(* POU Mio_GetCardMode, IL *)
(******************************************************************************
Description: Gets the mode of an IO-card.
Input:
  - CardId: ID of the card
Return: 
  - MIO_RETSTATE.RetCode: DINT => Success- or error code
  - MIO_RETSTATE.State: DWORD =>  Card mode (valid in case of success)
******************************************************************************)
FUNCTION Mio_GetCardMode : MIO_RETSTATE
VAR_INPUT
	CardId: DINT;
END_VAR
LD 0
END_FUNCTION

(* POU Mio_GetChanInf, IL *)
(******************************************************************************
Description: Gets information of an IO-channel of a card
Input:
  - CardId: ID of the card
  - Chan: Channel number
Return: 
  - MIO_RETCHANINF.RetCode: DINT => Success- or error-code
  - MIO_RETCHANINF.ChanCategory: DWORD =>  Channel-category (valid in case of success)
  - MIO_RETCHANINF.ChanFlags: DWORD =>  Properies of channel (valid in case of success)
******************************************************************************)
FUNCTION Mio_GetChanInf : MIO_RETCHANINF
VAR_INPUT
	CardId: DINT;
	Chan: DINT;
END_VAR
LD 0
END_FUNCTION

(* POU Mio_GetChanMode, IL *)
(******************************************************************************
Description: Gets the mode of a channel of an IO-card.
Input:
  - CardId: ID of the card
  - Chan: Channel number
Return: 
  - MIO_RETSTATE.RetCode: DINT => Success- or error-code
  - MIO_RETSTATE.State: DWORD =>  Channel mode (valid in case of success)
******************************************************************************)
FUNCTION Mio_GetChanMode : MIO_RETSTATE
VAR_INPUT
	CardId: DINT;
	Chan: DINT;
END_VAR
LD 0
END_FUNCTION

(* POU Mio_GetChanRangeInf, ST *)
(******************************************************************************
Description: Gets range information of an IO-channel of a card
Input:
  - CardId: ID of the card
  - Chan: Channel number
Return: 
  - MIO_RETCHANINF.RetCode: DINT => Success- or error-code
  - MIO_RETCHANINF.ChanCategory: DWORD =>  Channel-category (valid in case of success)
  - MIO_RETCHANINF.ChanFlags: DWORD =>  Properies of channel (valid in case of success)
******************************************************************************)
FUNCTION Mio_GetChanRangeInf : MIO_RETCHANRANGEINF
VAR_INPUT
	CardId: DINT;
	Chan: DINT;
END_VAR
;
END_FUNCTION

(* POU MIO_GetCustomerID, ST *)
FUNCTION_BLOCK MIO_GetCustomerID
VAR_INPUT
	Req : BOOL;
	CardId: DINT;
	CryptoKey: UDINT;
	AlgorithmId: UDINT;
	UserData: UDINT;
	CryptoFn: STRING(255);
END_VAR
VAR_OUTPUT
	Done : BOOL;
	Error : BOOL;
	Status : DINT;
	CustomerID: UDINT;
END_VAR
VAR
	Pltd : DWORD;
END_VAR
;
END_FUNCTION_BLOCK

(* POU Mio_GetError, IL *)
(******************************************************************************
Description: Gets the error state of a channel of an IO-card
Input:
  - CardId: ID of the card
  - Chan: Channel number
Return: 
  - MIO_RETSTATE.RetCode: DINT => Success- or error code
  - MIO_RETSTATE.State: DWORD =>  Error state (valid in case of success)
******************************************************************************)
FUNCTION Mio_GetError : MIO_RETSTATE
VAR_INPUT
	CardId: DINT;
	Chan: DINT;
END_VAR
LD 0
END_FUNCTION

(* POU Mio_GetExtCardInf, IL *)
(******************************************************************************
Description: Gets extended info for an IO-card
Input:
  - CardId: ID of the card
Return: 
  - MIO_RETEXTCARDINF.RetCode => Success- or error-code
  - MIO_RETEXTCARDINF.CardNb => Card number
  - MIO_RETEXTCARDINF.StationNb => Station number
  - MIO_RETEXTCARDINF.SlotNb => Slot number
  - MIO_RETEXTCARDINF.PreSlots => Precessing-also-used-slots
  - MIO_RETEXTCARDINF.PostSlots => Following-also-used-slots
  - MIO_RETEXTCARDINF.Mode => Mode of card driver
  - MIO_RETEXTCARDINF.State => State of Card-Driver
  - MIO_RETEXTCARDINF.CardType => Card type
  - MIO_RETEXTCARDINF.CardVariant => Card variant
  - MIO_RETEXTCARDINF.CardCategory => Card category
  - MIO_RETEXTCARDINF.CardFlags => Properties of card
  - MIO_RETEXTCARDINF.MaxChan => Number of channels
  - MIO_RETEXTCARDINF.Version => Card version
  - MIO_RETEXTCARDINF.DrvVersion => Necc. driver version
  - MIO_RETEXTCARDINF.Attribute => Defined/set attributes
  - MIO_RETEXTCARDINF.ProdTime => Date + time of production
  - MIO_RETEXTCARDINF.ProdNb => Serial no.-string
  - MIO_RETEXTCARDINF.Name => Name of card
  - MIO_RETEXTCARDINF.Info => Block of info text
  - MIO_RETEXTCARDINF.DrvName => Name of driver-*.M file
  - MIO_RETEXTCARDINF.Power => Power consumption in [mW]
  - MIO_RETEXTCARDINF.Current_5V => 5V Current sink/source in [mA]
  - MIO_RETEXTCARDINF.Current_P15V => +15V Current sink/source in [mA]
  - MIO_RETEXTCARDINF.Current_M15V => -15V Current sink/source in [mA]
  - MIO_RETEXTCARDINF.ModVerType => Version Type code
  - MIO_RETEXTCARDINF.RedundantRead => Redundant read of data if TRUE
  - MIO_RETEXTCARDINF.WriteVerify => Write verify of data if TRUE
  - MIO_RETEXTCARDINF.BusCheck => BUSCHECK supported if TRUE
  - MIO_RETEXTCARDINF.AliveCheck => ALIVECHECK supported if TRUE
  - MIO_RETEXTCARDINF.AssemblyCode => Function code lower part
  - MIO_RETEXTCARDINF.HwVariant => Hardware variant
  - MIO_RETEXTCARDINF.Reserved1 => Not used, 0 for now
  - MIO_RETEXTCARDINF.Settings => Flags that may be en-/disabled
  - MIO_RETEXTCARDINF.Fware => Firmware version
  - MIO_RETEXTCARDINF.ExStateInfo => Extended state information


******************************************************************************)
FUNCTION Mio_GetExtCardInf : MIO_RETEXTCARDINF
VAR_INPUT
	CardId: DINT;			(* use special value 16#80000001 for 'Cpu-Card' *)
END_VAR
	LD		0
END_FUNCTION

(* POU Mio_GetExtCardInf2, ST *)
(******************************************************************************
Description: Gets extended info for an IO-card
Input:
  - CardId: ID of the card
Return: 
  - MIO_RETEXTCARDINF2.RetCode => Success- or error-code
  - MIO_RETEXTCARDINF2.CardNb => Card number
  - MIO_RETEXTCARDINF2.StationNb => Station number
  - MIO_RETEXTCARDINF2.SlotNb => Slot number
  - MIO_RETEXTCARDINF2.PreSlots => Precessing-also-used-slots
  - MIO_RETEXTCARDINF2.PostSlots => Following-also-used-slots
  - MIO_RETEXTCARDINF2.Mode => Mode of card driver
  - MIO_RETEXTCARDINF2.State => State of Card-Driver
  - MIO_RETEXTCARDINF2.CardType => Card type
  - MIO_RETEXTCARDINF2.CardVariant => Card variant
  - MIO_RETEXTCARDINF2.CardCategory => Card category
  - MIO_RETEXTCARDINF2.CardFlags => Properties of card
  - MIO_RETEXTCARDINF2.MaxChan => Number of channels
  - MIO_RETEXTCARDINF2.Version => Card version
  - MIO_RETEXTCARDINF2.DrvVersion => Necc. driver version
  - MIO_RETEXTCARDINF2.Attribute => Defined/set attributes
  - MIO_RETEXTCARDINF2.ProdTime => Date + time of production
  - MIO_RETEXTCARDINF2.ProdNb => Serial no.-string
  - MIO_RETEXTCARDINF2.Name => Name of card
  - MIO_RETEXTCARDINF2.Info => Block of info text
  - MIO_RETEXTCARDINF2.DrvName => Name of driver-*.M file
  - MIO_RETEXTCARDINF2.Power => Power consumption in [mW]
  - MIO_RETEXTCARDINF2.Current_5V => 5V Current sink/source in [mA]
  - MIO_RETEXTCARDINF2.Current_P15V => +15V Current sink/source in [mA]
  - MIO_RETEXTCARDINF2.Current_M15V => -15V Current sink/source in [mA]
  - MIO_RETEXTCARDINF2.ModVerType => Version Type code
  - MIO_RETEXTCARDINF2.RedundantRead => Redundant read of data if TRUE
  - MIO_RETEXTCARDINF2.WriteVerify => Write verify of data if TRUE
  - MIO_RETEXTCARDINF2.BusCheck => BUSCHECK supported if TRUE
  - MIO_RETEXTCARDINF2.AliveCheck => ALIVECHECK supported if TRUE
  - MIO_RETEXTCARDINF2.AssemblyCode => Function code lower part
  - MIO_RETEXTCARDINF2.HwVariant => Hardware variant
  - MIO_RETEXTCARDINF2.Reserved1 => Not used, 0 for now
  - MIO_RETEXTCARDINF2.Settings => Flags that may be en-/disabled
  - MIO_RETEXTCARDINF2.ExStateInfo => Extended state information
  - MIO_RETEXTCARDINF2.Versions => Versions of this module (FW, Logic, ...)
  - MIO_RETEXTCARDINF2.PackageVers => Package version
  - MIO_RETEXTCARDINF2.PartNumber => Part number (0 if not available)
  - MIO_RETEXTCARDINF2.FirmBackup => Firmware can be recovered
  - MIO_RETEXTCARDINF2.Spare1 => Align it to 32 bit
  - MIO_RETEXTCARDINF2.Spare => Not used, 0 for now

******************************************************************************)
FUNCTION Mio_GetExtCardInf2 : MIO_RETEXTCARDINF2
VAR_INPUT
	CardId: DINT;			(* use special value 16#80000001 for 'Cpu-Card' *)
END_VAR
;
END_FUNCTION

(* POU Mio_GetIdToCard, IL *)
(******************************************************************************
Description: Gets the ID of an IO-card specified by card number
Input:
  - CardNum: Number of the card
Return: 
  - DINT => Pointer-ID of Card
  - In case of error: the special value -2147483648 (16#80000000) is returned
******************************************************************************)
FUNCTION Mio_GetIdToCard : DINT
VAR_INPUT
	CardNum : DINT;
END_VAR
LD 0
END_FUNCTION

(* POU Mio_GetInterruptInfo, ST *)
(******************************************************************************
Description: Returns informations regarding the current interrupt cycle(Is only
    valid if the current project is configured to be interrupt triggered-Event
    or Error interrupt.)
Input:
  - Dummy: 
Return: 
  -
******************************************************************************)
FUNCTION Mio_GetInterruptInfo : MIO_INTINFO
VAR_INPUT
	Dummy: DINT;
END_VAR
;
END_FUNCTION

(* POU Mio_GetNewSlaveReboot, ST *)
(******************************************************************************
Description: Returns the configuration for new FAST Bus slave stations behaviour.
Input:
  - Dummy: 
Return: 
  - TRUE: The controller will reboot, as soon as a new station is recognized.
  - FALSE: The new station will not be usable until a reboot happens. 
******************************************************************************)
FUNCTION Mio_GetNewSlaveReboot : BOOL
VAR_INPUT
	Dummy: DINT;
END_VAR
;
END_FUNCTION

(* POU Mio_GetNextError, IL *)
(******************************************************************************
Description: Finds the next IO-card / channel with an error state with attention to
Input:
  - StartCard:  Card to start the search from, valid range starts with -1 
  - StartChan:  Chan to start the search from, valid range starts with -1 
  - CardId: ID of the card
  - Chan: Channel number
Return: 
  - MIO_RETFOUND.RetCode: DINT => Success (0 or 1) - or error-code (<0)
  - MIO_RETFOUND.Card: DINT =>  Card with error (-1 for none)  (valid in case of success)
  - MIO_RETFOUND.Chan: DINT =>   Chan with error (-1 for none) (valid in case of success)
  - MIO_RETFOUND.State: DWORD =>  Error state (valid in case of success)
******************************************************************************)
FUNCTION Mio_GetNextError : MIO_RETFOUND
VAR_INPUT
	StartCard: DINT;		(* Card to start the search from, valid range starts with -1 *)
	StartChan: DINT;		(* Chan to start the search from, valid range starts with -1 *)
END_VAR
LD 0
END_FUNCTION

(* POU Mio_GetPackedValues, ST *)
(******************************************************************************
Description: Gets a number of packed values from IO-channels.
  Note:	Use Bit_Split to convert packed values into a BOOL array. 
        Due to more performance, process image channels aren't updated. 
		Don't use this function with a module in the process image configuration. 
Input:
  - CardId: ID of the card
  - StartAddr:  Address of bit buffer. 
  - StartChan:  First channel for reading (must be 1 or 17 or 33...).
  - ChannelCount:  Number of channels (must be 16 or 32 or 48....).
Output:
  - StartAddr:  Buffer filled with packed IO-bits. 
Return: 
  - DINT => Success- or error-code
******************************************************************************)
FUNCTION Mio_GetPackedValues : DINT
VAR_INPUT
	CardId: DINT;
	StartAddr: DWORD;
	StartChan: DWORD;
	ChannelCount: DWORD;
END_VAR
VAR
END_VAR
;
END_FUNCTION

(* POU Mio_GetScaleChanInf, ST *)
(******************************************************************************
Description: Get the scale ID of a channel.
Input:
  - CardId: Identifier CardId, result of Mio_GetIdToCard()
  - Chan:   Channel number (1 .. MaxChan)
Return: 
  - MIO_RETSCALEINF.Retcode   => Success- or error-code
	(MIO_ER_BADCHAN => channel does not exist;
	 MIO_ER_NOSCALEINF => channel is not scaled)
  - MIO_RETSCALEINF.pScaleinf => Scale-ID = Pointer to Scale information 
                                 of the channel
******************************************************************************)
FUNCTION Mio_GetScaleChanInf : MIO_RETSCALEINF
VAR_INPUT
	CardId	: DINT;		(* Card-Number *)
	Chan	: DINT;		(* Channel-Number *)
END_VAR
VAR
END_VAR
;
END_FUNCTION

(* POU Mio_GetScaledValueDINT, ST *)
(******************************************************************************
Description: Read the scaled value of a channel.
The channel has to be of scaling type SINT32, otherwise the call will fail with 
error code MIO_ER_WRONGFUNCTYPE.
Input:
  - CardId: Identifier CardId, result of Mio_GetIdToCard()
  - Chan:   Channel number (1 .. MaxChan)
Return: 
  - MIO_RETVALUE.RetCode: DINT => Success- or error-code
  - MIO_RETVALUE.Value:	  DINT => Scaled value (valid in case of success)
******************************************************************************)
FUNCTION Mio_GetScaledValueDINT  : MIO_RETVALUE
VAR_INPUT
	CardId	: DINT;
	Chan	: DINT;
END_VAR
VAR
END_VAR
;
END_FUNCTION

(* POU Mio_GetScaledValueLREAL, ST *)
(******************************************************************************
Description: Read the scaled value of a channel.
The channel has to be of scaling type REAL64, otherwise the call will fail with 
error code MIO_ER_WRONGFUNCTYPE.
Input:
  - CardId: Identifier CardId, result of Mio_GetIdToCard()
  - Chan:   Channel number (1 .. MaxChan)
Return: 
  - MIO_RETVALUE.RetCode: DINT => Success- or error-code
  - MIO_RETVALUE.Value:	  DINT => Scaled value (valid in case of success)
******************************************************************************)
FUNCTION Mio_GetScaledValueLREAL : MIO_RETVALUE_LREAL
VAR_INPUT
	CardId	: DINT;
	Chan	: DINT;
END_VAR
VAR
END_VAR
;
END_FUNCTION

(* POU Mio_GetSelect, IL *)
(******************************************************************************
Description: Gets the SelectInfo of an IO card's channel
Input:
  - CardId: ID of the card
  - Chan: Channel number
Return: 
  - MIO_RETSTATE.RetCode: DINT => Success- or error code
  - MIO_RETSTATE.State: DWORD =>  Select info (valid in case of success)
******************************************************************************)
FUNCTION Mio_GetSelect : MIO_RETSTATE
VAR_INPUT
	CardId: DINT;
	Chan: DINT;
END_VAR
LD 0
END_FUNCTION

(* POU Mio_GetValue, IL *)
(******************************************************************************
Description: Gets the value of an IO-channel 
Input:
  - CardId: ID of the card
  - Chan: Channel number
Return: 
  - MIO_RETVALUE.RetCode: DINT => Success- or error-code
  - MIO_RETVALUE.Value: DINT =>  IO-value (valid in case of success)
******************************************************************************)
FUNCTION Mio_GetValue : MIO_RETVALUE
VAR_INPUT
	CardId: DINT;
	Chan: DINT;
END_VAR
	LD		0
END_FUNCTION

(* POU Mio_GetValues, IL *)
(******************************************************************************
Description: Gets a number of values from IO-channels
Input:
  - CardId: ID of the card
  - StartAddr:  Must be the address of the first DINT/UDINT-value 
  - EndAddr:  Must be the address of the last DINT/UDINT-value 
  - NumberOf:  [StartAddr..EndAddr] must contain number of - values 
Return: 
  - DINT => Success- or Error-Code
******************************************************************************)
FUNCTION Mio_GetValues : DINT
VAR_INPUT
	CardId: DINT;
	StartAddr: DWORD;		(* Must be the address of the first DINT/UDINT-value *)
	EndAddr: DWORD; 		(* Must be the address of the last DINT/UDINT-value *)
	NumberOf: DINT; 		(* [StartAddr..EndAddr] must contain number of - values *)
END_VAR
LD 0
END_FUNCTION

(* POU Mio_GetVersion, ST *)
(******************************************************************************
Description: Returns the version string of the library. In simulation always
	'' is returned.

Input:
	- dummy

Return: 
	Version string
******************************************************************************)
FUNCTION Mio_GetVersion : STRING(15)
VAR_INPUT
	dummy:		BOOL;
END_VAR
VAR
END_VAR
Mio_GetVersion := '';
END_FUNCTION

(* POU Mio_Reset, IL *)
(******************************************************************************
Description: Resets an IO-Card
Input:
  - CardId: ID of the card
Return: 
  - DINT => Success- or error code
******************************************************************************)
FUNCTION Mio_Reset : DINT
VAR_INPUT
	CardId: DINT;
END_VAR
LD 0
END_FUNCTION

(* POU Mio_SetBadSlaveReboot, ST *)
(******************************************************************************
Description: Changes the behaviour for bad FAST Bus slave stations.
Input:
  - BadSlaveReboot: 
Return: 
  - TRUE: The return value ist TRUE, if the functionality is supported
    (MSys >= V1.06). See also Mio_GetBadSlaveReboot(FUN).
  - FALSE: 
******************************************************************************)
FUNCTION Mio_SetBadSlaveReboot : BOOL
VAR_INPUT
	BadSlaveReboot : BOOL;
END_VAR
;
END_FUNCTION

(* POU Mio_SetBlk, IL *)
(******************************************************************************
Description: Writes a block value of a IO-channel
Input:
  - CardId: ID of the card
  - Chan: Channel number
  - pValue: Pointer to buffer which holds the data to write
  - Len: Amount of bytes to be written
Output:
Return: 
  - RetCode: DINT => Success- or error-code
******************************************************************************)
FUNCTION Mio_SetBlk : DINT
VAR_INPUT
	CardId: DINT;
	Chan: DINT;
	pValue: POINTER TO BYTE;
	Len: UDINT;
END_VAR
LD 0
END_FUNCTION

(* POU Mio_SetCardMode, IL *)
(******************************************************************************
Description: Sets the Card Mode of an IO Card
Input:
  - CardId: ID of the card
  - Mode:  Card mode to be set 
Return: 
  - DINT => Success- or error code
******************************************************************************)
FUNCTION Mio_SetCardMode : DINT
VAR_INPUT
	CardId: DINT;
	Mode: DWORD;	(* Card mode to be set *)
END_VAR
LD 0
END_FUNCTION

(* POU Mio_SetChanMode, IL *)
(******************************************************************************
Description: Sets the channel mode of an IO-card's channel
Input:
  - CardId: ID of the card
  - Chan: Channel number
  - Mode:  Chan mode to be set 
Return: 
  - DINT => Success- or error code
******************************************************************************)
FUNCTION Mio_SetChanMode : DINT
VAR_INPUT
	CardId: DINT;
	Chan: DINT;
	Mode: DWORD;	(* Chan-Mode to be set *)
END_VAR
LD 0
END_FUNCTION

(* POU Mio_SetNewSlaveReboot, ST *)
(******************************************************************************
Description: Changes the behaviour for New FAST-Bus slave stations.
Input:
  - NewSlaveReboot: 
Return: 
  - TRUE: The return value ist TRUE, if the functionality is supported
    (MSys >= V1.06). See also Mio_GetNewSlaveReboot(FUN). 
  - FALSE: 
******************************************************************************)
FUNCTION Mio_SetNewSlaveReboot : BOOL
VAR_INPUT
	NewSlaveReboot : BOOL;
END_VAR
;
END_FUNCTION

(* POU Mio_SetPackedValues, ST *)
(******************************************************************************
Description: Sets a number of packed values to IO-channels.
  Note:	Use Bit_Pack to pack values from an BOOL array. 
		Due to more performance, process image channels aren't updated. 
		Don't use this function with a module in the process image configuration. 
Input:
  - CardId: ID of the card
  - StartAddr:  Address of bit buffer 
  - StartChan:  First channel for writing (must be 1 or 17 or 33...).
  - ChannelCount:  Number of channels (must be 16 or 32 or 48....).
Return: 
  - DINT => Success- or error-code
******************************************************************************)
FUNCTION Mio_SetPackedValues : DINT
VAR_INPUT
	CardId: DINT;
	StartAddr: DWORD;
	StartChan: DWORD;
	ChannelCount: DWORD;
END_VAR
VAR
END_VAR
;
END_FUNCTION

(* POU Mio_SetScaledValueDINT, ST *)
(******************************************************************************
Description: Write a scaled value.
The channel has to be of scaling type SINT32, otherwise the call will fail with 
error code MIO_ER_WRONGFUNCTYPE.
The process image is not updated by a call to this function.
Input:
  - CardId: Identifier CardId, result of Mio_GetIdToCard()
  - Chan:   Channel number (1 .. MaxChan)
  - Value:  Scaled value to be set
Return: 
  - DINT => Success- or error-code
******************************************************************************)
FUNCTION Mio_SetScaledValueDINT : DINT
VAR_INPUT
	CardId	: DINT;
	Chan	: DINT;
	Value	: DINT;		(* Value to be set *)
END_VAR
VAR
END_VAR
;
END_FUNCTION

(* POU Mio_SetScaledValueLREAL, ST *)
(******************************************************************************
Description: Write a scaled value.
The channel has to be of scaling type REAL64, otherwise the call will fail with 
error code MIO_ER_WRONGFUNCTYPE.
The process image is not updated by a call to this function.
Input:
  - CardId: Identifier CardId, result of Mio_GetIdToCard()
  - Chan:   Channel number (1 .. MaxChan)
  - Value:  Scaled value to be set
Return: 
  - DINT => Success- or error-code
******************************************************************************)
FUNCTION Mio_SetScaledValueLREAL : DINT
VAR_INPUT
	CardId	: DINT;
	Chan	: DINT;
	Value	: LREAL;		(* Value to be set *)
END_VAR
VAR
END_VAR
;
END_FUNCTION

(* POU Mio_SetSelect, IL *)
(******************************************************************************
Description: Sets the select info of an IO card's channel
Input:
  - CardId: ID of the card
  - Chan: Channel number
  - Select:  Selection info to be applied 
Return: 
  -
******************************************************************************)
FUNCTION Mio_SetSelect : DINT
VAR_INPUT
	CardId: DINT;
	Chan: DINT;
	Select: DWORD;	(* Selection info to be applied *)
END_VAR
LD 0
END_FUNCTION

(* POU Mio_SetValue, IL *)
(******************************************************************************
Description: Sets the value of an IO-channel
Input:
  - CardId: Must be the address
  - Chan: Channel number
  - Value:  Value to be set 
Return: 
  - DINT => Success- or error-code
******************************************************************************)
FUNCTION Mio_SetValue : DINT
VAR_INPUT
	CardId: DINT;
	Chan: DINT;
	Value: DINT;		(* Value to be set *)
END_VAR
LD 0
END_FUNCTION

(* POU Mio_SetValues, IL *)
(******************************************************************************
Description: Sets a number of values to IO-card channels.
Input:
  - CardId: Must be the address
  - StartAddr:  Must be the address of the first DINT/UDINT value 
  - EndAddr:  Must be the address of the last DINT/UDINT value 
  - NumberOf:  [StartAddr..EndAddr] must contain number of - values 
Return: 
  - DINT => Success- or error code
******************************************************************************)
FUNCTION Mio_SetValues : DINT
VAR_INPUT
	CardId: DINT;
	StartAddr: DWORD;		(* Must be the address of the first DINT/UDINT value *)
	EndAddr: DWORD; 		(* Must be the address of the last DINT/UDINT value *)
	NumberOf: DINT; 		(* [StartAddr..EndAddr] must contain number of values *)
END_VAR
LD 0
END_FUNCTION

(* POU MIO_TestCustomerID, ST *)
FUNCTION_BLOCK MIO_TestCustomerID
VAR_INPUT
	Req : BOOL;
	CryptoKey: UDINT;
	CustomerID: UDINT;
	Range: UDINT;
	AlgorithmId: UDINT;
	UserData: UDINT;
	CryptoFn: STRING(255);
	PrintMsg: BOOL;
END_VAR
VAR_OUTPUT
	Done : BOOL;
	Error : BOOL;
	Status : DINT;
END_VAR
VAR
	Pltd : DWORD;
END_VAR
;
END_FUNCTION_BLOCK
